Fanuc KAREL source: XML_SETVAR.kl

PROGRAM T
%NOLOCKGROUP
VAR
 v0 : FILE
 v1 : STRING[40]
 v2 : STRING[40]
 v3 : INTEGER
BEGIN
 XML_SETVAR(v0, v1, v2, v3)
END T
